{attribute addProperty BoxType "EL2911-0000-0016"}
{attribute addProperty Id "OutputsOutputs_BAABD9C981"}
{attribute addProperty CRC "1237327669"}
{attribute addProperty SizeInBites "8"}
{attribute addProperty SizeInBytes "1"}
TYPE Module_2_FSOUT_49C01F35 :
STRUCT
	{attribute addProperty Name "Outputs"}
	Outputs  : Outputs_BAABD9C9;
END_STRUCT
END_TYPE

(* stored: Version 1.2.0.0, ProductVersion 3.1.4024.9
   DUT Module_2_FSOUT_49C01F35: Id {b9f2cad4-1668-4951-be0a-a7c5865964d0} *)
